Staubli VAL3: Control_PanelXY.pgx

public program Control_PanelXY(num x_nPanelLTopX, num x_nPanelLTopY, num x_nPanelWidthX, num x_nPanelLengthY)
begin

  //对于新建的框和列表进行位置和大小的设定

  //对于数值范围进行判断，一般的情况可以使用min,max就可以
  //如果传入的参数不正确，则设定初始值
  nPanelLTopX=min(max(0,x_nPanelLTopX),38)
  nPanelLTopY=min(max(0,x_nPanelLTopY),12)

  nPanelWidthX=min(max(0,x_nPanelWidthX),38)
  nPanelLengthY=min(max(0,x_nPanelLengthY),12)


end
